# EPICS autosave request: iocs/motion/req/motion_settings.req
# Operator settings restored across IOC restarts.
# The target position is deliberately NOT saved — restoring it would
# command a move on IOC restart.
$(P):M1:VELO
